Fanuc KAREL source: kd00036.KL

-- PROVISIONAL review KL for V940-1; original PC SHA256 ef0f3f5593cf93c945ab665c554743569a8b07df8815edd03745b3460e177426
-- Incomplete behavior may be omitted. Consult companion uncertainty JSON. Do not deploy.
PROGRAM KD00036
%NOLOCKGROUP
VAR
  I : INTEGER
  J : INTEGER
  B : BOOLEAN
  R : REAL
  S : STRING[80]
BEGIN
  -- V9_ZERO_TABLE_METADATA_HINT layout=0001; no indexed target words; source/name/runtime held
  -- UNRESOLVED_PC offsets 5-17; opcodes 9D,81,18,9D,1B,9D,12,13,04
  -- UNRESOLVED_PC offsets 22-26; opcodes 7F
END KD00036
